SUBAPPLICATION OPC_PUB_EX_1 (* Subapplication Type *)
  (* Standard: 61499-2 *)
  (* Version 1.0, 2022-03-09, Maximilian Scharf *)
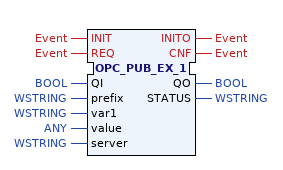
  EVENT_INPUT
    INIT;
    REQ;
  END_EVENT
  EVENT_OUTPUT
    INITO;
    CNF;
  END_EVENT
  VAR_INPUT
    QI : BOOL;
    prefix : WSTRING;
    var1 : WSTRING := STRING#'a';
    value : ANY;
    server : WSTRING;
  END_VAR
  VAR_OUTPUT
    QO : BOOL;
    STATUS : WSTRING;
  END_VAR
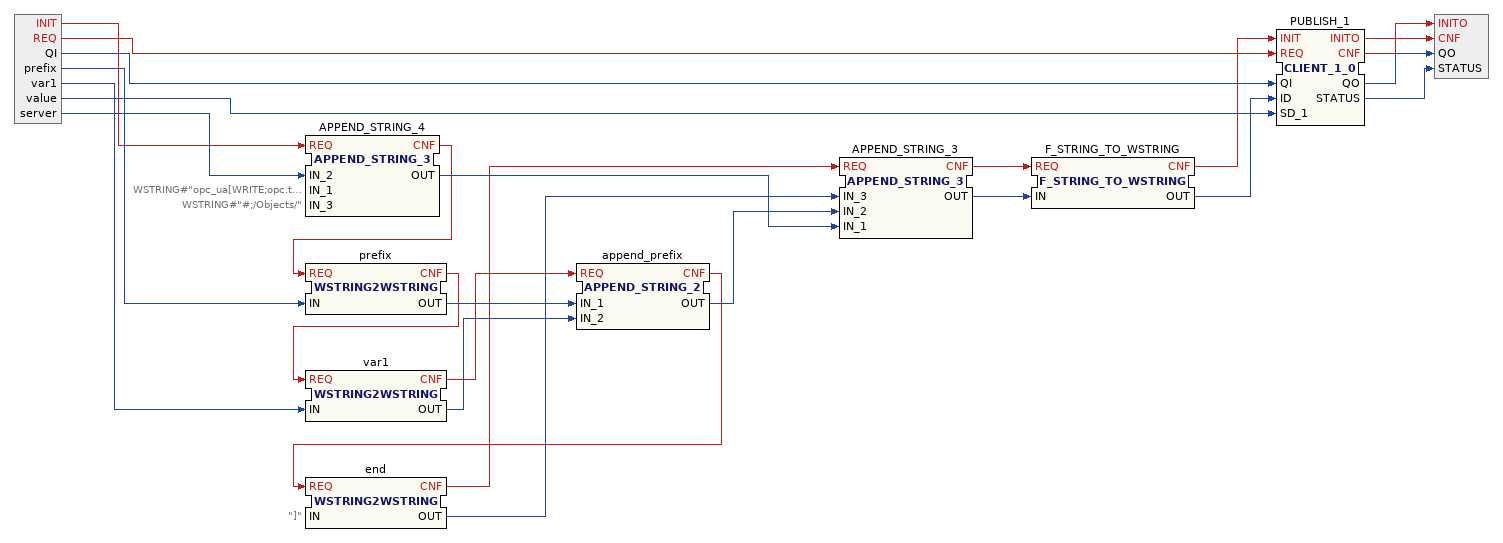
  FBS
    F_STRING_TO_WSTRING : F_STRING_TO_WSTRING;
    APPEND_STRING_3 : APPEND_STRING_3;
    end : WSTRING2WSTRING(IN := "]");
    var1 : WSTRING2WSTRING;
    prefix : WSTRING2WSTRING;
    append_prefix : APPEND_STRING_2;
    APPEND_STRING_4 : APPEND_STRING_3(IN_1 := WSTRING#"opc_ua[WRITE;opc.tcp://", IN_3 := WSTRING#"#;/Objects/");
    PUBLISH_1 : CLIENT_1_0;
  END_FBS
  EVENT_CONNECTIONS
    APPEND_STRING_3.CNF TO F_STRING_TO_WSTRING.REQ;
    prefix.CNF TO var1.REQ;
    var1.CNF TO append_prefix.REQ;
    append_prefix.CNF TO end.REQ;
    end.CNF TO APPEND_STRING_3.REQ;
    APPEND_STRING_4.CNF TO prefix.REQ;
    INIT TO APPEND_STRING_4.REQ;
    F_STRING_TO_WSTRING.CNF TO PUBLISH_1.INIT;
    REQ TO PUBLISH_1.REQ;
    PUBLISH_1.INITO TO INITO;
    PUBLISH_1.CNF TO CNF;
  END_CONNECTIONS
  DATA_CONNECTIONS
    APPEND_STRING_3.OUT TO F_STRING_TO_WSTRING.IN;
    end.OUT TO APPEND_STRING_3.IN_3;
    var1 TO var1.IN;
    prefix TO prefix.IN;
    prefix.OUT TO append_prefix.IN_1;
    var1.OUT TO append_prefix.IN_2;
    append_prefix.OUT TO APPEND_STRING_3.IN_2;
    APPEND_STRING_4.OUT TO APPEND_STRING_3.IN_1;
    server TO APPEND_STRING_4.IN_2;
    QI TO PUBLISH_1.QI;
    F_STRING_TO_WSTRING.OUT TO PUBLISH_1.ID;
    value TO PUBLISH_1.SD_1;
    PUBLISH_1.QO TO QO;
    PUBLISH_1.STATUS TO STATUS;
  END_CONNECTIONS
END_SUBAPPLICATION
